(* IEC 61131-3 sources: test/Class/HmiImageList, 1 file *)

(* ---- HmiImageList.st ---- *)
(*!
<Class
	Name               = "HmiImageList"
	Revision           = "0.3"
	RealtimeTask       = "false"
	CyclicTask         = "false"
	BackgroundTask     = "false"
	Sigmatek           = "true"
	OSInterface        = "false"
	HighPriority       = "false"
	Automatic          = "false"
	UpdateMode         = "Prescan"
	SharedCommandTable = "true"
	Objectsize         = "(284,120)">
	<Channels>
		<Client Name="Label" Required="true" Internal="true"/>
		<Client Name="StringLib" Required="true" Internal="false"/>
	</Channels>
	<Dependencies>
		<Files>
			<File Path=".\Class\HmiImageList\CBmpConv.cpp"/>
			<File Path=".\Class\HmiImageList\CBmpConv.h" Include="false"/>
		</Files>
	</Dependencies>
	<RevDoku>
		<Owner Company="sigmatek" Author="kolott"/>
		<Dokumentation Revision="0.3" Date="2018-03-06" Author="kolott" Company="sigmatek" Description="sa40364, DEVSW-395: New method XChange() to xchange image done with lse by Bitmap"/>
		<Dokumentation Revision="0.2" Date="2014-04-15" Author="kolott" Company="sigmatek" Description="new method FreeMem()"/>
		<Dokumentation Revision="0.1" Date="2014-02-28" Author="kolott" Company="sigmatek" Description="betterment speed"/>
	</RevDoku>
	<Network Name="HmiImageList">
		<!-- List of Components in this network -->
		<Components>
			<Object
				Name       = "_base"
				Class      = "HmiBaseList"
				Position   = "(218,120)"
				Visualized = "false">
				<Channels>
					<Server Name="ClassSvr"/>
					<Client Name="File"/>
				</Channels>
			</Object>
			<Object
				Name       = "Label"
				Class      = "HmiAsciiBuffer"
				Position   = "(210,300)"
				Visualized = "false">
				<Channels>
					<Server Name="ClassSvr"/>
					<Client Name="File"/>
					<Client Name="StringLib"/>
				</Channels>
			</Object>
		</Components>
		<Comments>
		</Comments>
		<!-- List of Connections in this network -->
		<Connections>
			<Connection Source="this.ClassSvr" Destination="_base.ClassSvr" Vertices="(690,210),(518,210),"/>
			<Connection Source="_base.File" Destination="this.File" Vertices="(218,210),(38,210),"/>
			<Connection Source="this.Label" Destination="Label.ClassSvr"/>
			<Connection Source="Label.File" Destination="this.File" Vertices="(210,390),(38,210),"/>
			<Connection Source="Label.StringLib" Destination="this.StringLib" Vertices="(210,450),(38,270),"/>
		</Connections>
		<!-- Headerfiles -->
		<Options>
		</Options>
	</Network>
</Class>
*)
#pragma using HmiBaseList

HmiImageList : CLASS
: HmiBaseList
  //Servers:
  //Clients:
	Label 	: CltChCmd_HmiAsciiBuffer;
	StringLib 	: CltChCmd_HmiStrLib;
  //Variables:
		No 	: UDINT;
		Ptr 	: ^HMI_IMAGEINFO;
		IncNo 	: UDINT;
  //Functions:

	FUNCTION HmiImageList
		VAR_OUTPUT
			ret_code 	: ConfStates;
		END_VAR;

	FUNCTION VIRTUAL Load
		VAR_OUTPUT
			retcode 	: BOOL;
		END_VAR;

	FUNCTION VIRTUAL Free;

	FUNCTION Init_IMAGE
		VAR_INPUT
			pi 	: ^HMI_IMAGEINFO;
		END_VAR;

	FUNCTION Free_IMAGE
		VAR_INPUT
			pi 	: ^HMI_IMAGEINFO;
		END_VAR;

	FUNCTION GLOBAL Get
		VAR_INPUT
			index 	: UDINT;
		END_VAR
		VAR_OUTPUT
			retcode 	: ^HMI_IMAGEINFO;
		END_VAR;

	FUNCTION GLOBAL IncNumber
		VAR_OUTPUT
			retcode 	: UDINT;
		END_VAR;

	FUNCTION GLOBAL GetIndexByName
		VAR_INPUT
			name 	: ^CHAR;
		END_VAR
		VAR_OUTPUT
			retcode 	: UDINT;
		END_VAR;

	FUNCTION GLOBAL FreeMem;

	FUNCTION GLOBAL XChange
		VAR_INPUT
			name 	: ^CHAR;
			dpne 	: ^CHAR;
		END_VAR
		VAR_OUTPUT
			retcode 	: BOOL;
		END_VAR;
  //Tables:
	FUNCTION @STD
		VAR_OUTPUT
			ret_code	: CONFSTATES;
		END_VAR;
	FUNCTION GLOBAL TAB @CT_;
END_CLASS;

#pragma using HmiAsciiBuffer
#pragma usingLtd HmiStrLib

#include "CBmpConv.h"

FUNCTION HmiImageList::HmiImageList
	VAR_OUTPUT
		ret_code 	: ConfStates;
	END_VAR

  Ptr      := NIL;
  No       := 0;
  IncNo    := 0;
	ret_code := C_OK;
  ClassSvr := 0;

END_FUNCTION

FUNCTION HmiImageList::Init_IMAGE
	VAR_INPUT
		pi 	: ^HMI_IMAGEINFO;
	END_VAR

  pi^.width       := 0;
  pi^.height      := 0;
  pi^.transparent := 0;
  pi^.state       := 0;
  pi^.datano      := 0;
  pi^.ptr         := NIL;
  pi^.index35     := HMI_DEFSCOPE;

END_FUNCTION

FUNCTION HmiImageList::Free_IMAGE
	VAR_INPUT
		pi 	: ^HMI_IMAGEINFO;
	END_VAR

  File.Memory(#pi^.ptr, 0);
  Init_IMAGE(pi);

END_FUNCTION

FUNCTION VIRTUAL HmiImageList::Free
  VAR
  	ph : ^HMI_IMAGEINFO;
  END_VAR

  ph := Ptr;
  while(No) do
    Free_IMAGE(ph);
    No -= 1;
    ph += sizeof(HMI_IMAGEINFO);
  end_while;

  if(Ptr <> NIL) then
    File.Memory(#Ptr$^void, 0);
  end_if;
  Label.Free();
  Ptr      := NIL;
  No       := 0;
  IncNo    := 0;
  ClassSvr := 0;

END_FUNCTION

FUNCTION VIRTUAL HmiImageList::Load
	VAR_OUTPUT
		retcode 	: BOOL;
	END_VAR
  var
    anz : uint;
    tmp : ^HMI_IMAGEINFO;
    single : uint;
    size : udint;
  end_var;

  retcode := false;

  if(File.FRead(#single$void, 2) = true) then
    if(single = 0) then // kein singleimagefileformat
      File.FRead(#anz$void, 2);
      if(File.FMemory(#Ptr$^void, anz * sizeof(HMI_IMAGEINFO)) = true) then
        tmp := Ptr;
        while(anz) do
          Init_IMAGE(tmp);

          File.FRead(#tmp^.datano$void, 4);
          File.FRead(#tmp^.width$void, 2);
          File.FRead(#tmp^.height$void, 2);
          File.FRead(#tmp^.transparent$void, 2);
          File.FRead(#tmp^.state$void, 2);

          if(tmp^.state and 0x0008) then // 8bit farbinfo
            size := tmp^.datano * 2;
            if(File.FMemory(#tmp^.ptr, size) = true) then
              File.FRead(tmp^.ptr, size);
            end_if;
          else
            size := tmp^.datano * 3;
            if(File.FMemory(#tmp^.ptr, size) = true) then
              File.FRead(tmp^.ptr, size);
            end_if;
          end_if;

          anz -= 1;
          No  += 1;
          tmp += sizeof(HMI_IMAGEINFO);
        end_while;

        if(File.FChkFile() = true) then
          Label.Load();
          retcode := true;
        else
          Free();
        end_if;
      end_if;
    end_if;
  end_if;

  ClassSvr := to_dint(No);

END_FUNCTION

FUNCTION GLOBAL HmiImageList::Get
	VAR_INPUT
		index 	: UDINT;
	END_VAR
	VAR_OUTPUT
		retcode 	: ^HMI_IMAGEINFO;
	END_VAR

  retcode := NIL;
  if(index < No) then
    retcode := Ptr + (index * sizeof(HMI_IMAGEINFO));
  end_if;

END_FUNCTION

FUNCTION GLOBAL HmiImageList::GetIndexByName
	VAR_INPUT
		name 	: ^CHAR;
	END_VAR
	VAR_OUTPUT
		retcode 	: UDINT;
	END_VAR

  retcode := Label.GetNoByName(name);

END_FUNCTION

FUNCTION GLOBAL HmiImageList::IncNumber
	VAR_OUTPUT
		retcode 	: UDINT;
	END_VAR

  retcode := IncNo;
  IncNo += 1;

END_FUNCTION

FUNCTION GLOBAL HmiImageList::FreeMem

  Free();

END_FUNCTION

FUNCTION GLOBAL HmiImageList::XChange
	VAR_INPUT
		name 	: ^CHAR;
		dpne 	: ^CHAR;
	END_VAR
	VAR_OUTPUT
		retcode 	: BOOL;
	END_VAR
  VAR
  	pdst : ^HMI_IMAGEINFO;
    pbmp : ^void;
    praw, traw : ^tcRaw;
    pbmo : ^tcBmo;
  END_VAR

  retcode := false;

  if((name <> NIL) & (dpne <> NIL)) then

    pdst := Get(GetIndexByName(name)); // pointer auf dst ermitteln
    if(pdst <> NIL) then

      pbmp := File.GetFileContent(dpne); // file auslesen
      if(pbmp <> NIL) then
          praw := bcBitmapToRaw(pbmp); // in raw format konvertieren
          File.FMemory(#pbmp, 0); // free filecontent, wird nicht mehr benötigt

          if(praw <> NIL) then
            if((praw^.width <> pdst^.width) | (praw^.height <> pdst^.height)) then
              traw := bcRawClone(pdst^.width, pdst^.height, praw); // grösse ändern
              if(traw <> NIL) then
                bcFreeRaw(praw);
                praw := traw;
              end_if;
            end_if;

            pbmo := bcRawToBmo(praw); // in bmo-format wandeln
            if(pbmo <> NIL) then

              pdst^.width       := pbmo^.width;
              pdst^.height      := pbmo^.height;
              pdst^.datano      := pbmo^.datano;
              pdst^.transparent := pbmo^.transparent;
              pdst^.datano      := pbmo^.datano;
              pdst^.state       := pbmo^.state;

              File.FMemory(#pdst^.ptr, 0); // alten bmo-puffer freigeben
              pdst^.ptr         := pbmo^.ptr;
              pbmo^.ptr         := NIL; // bmp pointer initialisieren

              bcFreeBmo(pbmo); // bmo freigeben
              retcode := true;
            end_if;

            bcFreeRaw(praw); // free praw

          end_if;

        File.FMemory(#pbmp, 0); // ggf. free filecontent
      end_if;
    end_if;
  end_if;

END_FUNCTION
